(* IEC 61131-3 sources: AXOpen/src/showcase/app/src/ComponentsRexrothDrives/Documentation, 1 file *)

(* ---- Component_1.st ---- *)
USING AXOpen.Components.Abstractions.Drives;
USING AXOpen.Core;

NAMESPACE AXOpen.Components.Rexroth.Drives
    {S7.extern=ReadWrite}
    CLASS Component_1 EXTENDS AXOpen.Core.AxoObject
        //<ComponentDeclaration>
        VAR PUBLIC
            IndraDrive : AXOpen.Components.Rexroth.Drives.AxoIndraDrive;
        END_VAR
        //</ComponentDeclaration>

        //<InitializationArgumentsDeclaration>
        VAR PUBLIC
            manualControl   :   BOOL;
            Enable          :   BOOL;                       //  As long as ‘Enable’ is true, power is being enabled.
            EnablePositive  :   BOOL;                       //  As long as ‘Enable’ is true, this permits motion in positive direction
            EnableNegative  :   BOOL;                       //  As long as ‘Enable’ is true, this permits motion in negative direction
        END_VAR
        //</InitializationArgumentsDeclaration>

        METHOD PUBLIC OVERRIDE Run
            VAR_INPUT
                inParent : IAxoObject;
            END_VAR

            SUPER.Run(inParent);

            IF(manualControl) THEN
                IndraDrive.ActivateManualControl();
            END_IF;
            //<Initialization>
            IndraDrive.Run(inParent               :=  THIS,
                            hwID                :=  AXOpen.Showcase.HwIdentifiers#rexroth_indradrive_HwID,
                            Enable              :=  Enable,
                            EnablePositive      :=  EnablePositive,
                            EnableNegative      :=  EnableNegative);
            //</Initialization>

        THIS.UseInSequencer();
        END_METHOD

        //<Usage>
        VAR PUBLIC
            Sequencer : AxoSequencer;
            Steps : ARRAY[0..30] OF AXOpen.Core.AxoStep;
        END_VAR

        VAR PRIVATE
            _Valid : BOOL;
            _BoolValue  : BOOL;
            _DintValue  : DINT;
            _RealValue  : REAL;
            _i          : INT;
        END_VAR
        METHOD PRIVATE UseInSequencer

            Sequencer.Run(THIS);
            Sequencer.Open();
            Sequencer.SequenceMode := eAxoSequenceMode#RunOnce;

            _i := 0;
            IF(Steps[_i].Execute(Sequencer, 'Restore')) THEN
                manualControl := FALSE;
                Enable := FALSE;
                EnablePositive := FALSE;
                EnableNegative := FALSE;
                IndraDrive.Restore();
                Sequencer.MoveNext();
            END_IF;

            _i := _i + 1;
            IF(Steps[_i].Execute(Sequencer, 'Reset drive')) THEN
                IF(IndraDrive.AxoReset().IsDone()) THEN
                    Sequencer.MoveNext();
                END_IF;
            END_IF;

            _i := _i + 1;
            IF(Steps[_i].Execute(Sequencer, 'Enable drive')) THEN
                Enable := TRUE;
                EnablePositive := TRUE;
                EnableNegative := TRUE;
                IF(IndraDrive.AxoPower_Status) THEN
                    Sequencer.MoveNext();
                END_IF;
            END_IF;

            _i := _i + 1;
            IF(Steps[_i].Execute(Sequencer, 'Drive homming')) THEN
                IF(IndraDrive.AxoHome(  Position        :=  LREAL#5.0,
                                            HommingMode     :=  INT#551,
                                            Velocity        :=  LREAL#1.0,
                                            Acceleration    :=  LREAL#50.0,
                                            Deceleration    :=  LREAL#50.0
                                            ).IsDone()) THEN
                    IndraDrive.Restore();
                    Sequencer.MoveNext();
                END_IF;
            END_IF;

            _i := _i + 1;
            IF(Steps[_i].Execute(Sequencer, 'Check position')) THEN
                IF(IndraDrive.ActualPosition >=4.9 AND  IndraDrive.ActualPosition <=5.1) THEN
                    Sequencer.MoveNext();
                END_IF;
            END_IF;

            _i := _i + 1;
            IF(Steps[_i].Execute(Sequencer, 'Set position')) THEN
                IF(IndraDrive.AxoSetPosition(Position :=  LREAL#0.0).IsDone()) THEN
                    IndraDrive.Restore();
                    Sequencer.MoveNext();
                END_IF;
            END_IF;

            _i := _i + 1;
            IF(Steps[_i].Execute(Sequencer, 'Check position')) THEN
                IF(IndraDrive.ActualPosition >=-0.1 AND  IndraDrive.ActualPosition <=0.1) THEN
                    Sequencer.MoveNext();
                END_IF;
            END_IF;

            _i := _i + 1;
            IF(Steps[_i].Execute(Sequencer, 'Move absolute')) THEN
                IF(IndraDrive.AxoMoveAbsolute(  Position        :=  LREAL#5.0,
                                                    Velocity        :=  LREAL#10.0,
                                                    Acceleration    :=  LREAL#50.0,
                                                    Deceleration    :=  LREAL#50.0,
                                                    Jerk            :=  LREAL#50.0
                                                    ).IsDone()) THEN
                    IndraDrive.Restore();
                    Sequencer.MoveNext();
                END_IF;
            END_IF;

            _i := _i + 1;
            IF(Steps[_i].Execute(Sequencer, 'Check position')) THEN
                IF(IndraDrive.ActualPosition >=4.9 AND  IndraDrive.ActualPosition <=5.1) THEN
                    Sequencer.MoveNext();
                END_IF;
            END_IF;

            _i := _i + 1;
            IF(Steps[_i].Execute(Sequencer, 'Move additive')) THEN
                IndraDrive.AxoMoveAbsolute(  Position           :=  LREAL#10.0,
                                                    Velocity        :=  LREAL#1.0,
                                                    Acceleration    :=  LREAL#50.0,
                                                    Deceleration    :=  LREAL#50.0,
                                                    Jerk            :=  LREAL#50.0
                                                    );
                IF IndraDrive.ActualPosition > 7.5 THEN
                    IndraDrive.AxoMoveAdditive(  Distance        :=  LREAL#5.0,
                                                        Velocity        :=  LREAL#5.0,
                                                        Acceleration    :=  LREAL#50.0,
                                                        Deceleration    :=  LREAL#50.0,
                                                        Jerk            :=  LREAL#50.0
                                                        );
                END_IF;
                IF(IndraDrive.AxoMoveAdditive_Task.IsDone()) THEN
                    IndraDrive.Restore();
                    Sequencer.MoveNext();
                END_IF;
            END_IF;

            _i := _i + 1;
            IF(Steps[_i].Execute(Sequencer, 'Check position')) THEN
                IF(IndraDrive.ActualPosition >=14.9 AND  IndraDrive.ActualPosition <=15.1) THEN
                    Sequencer.MoveNext();
                END_IF;
            END_IF;

            _i := _i + 1;
            IF(Steps[_i].Execute(Sequencer, 'Move relative')) THEN
                IF(IndraDrive.AxoMoveRelative(  Distance        :=  LREAL#-5.0,
                                                    Velocity        :=  LREAL#10.0,
                                                    Acceleration    :=  LREAL#50.0,
                                                    Deceleration    :=  LREAL#50.0,
                                                    Jerk            :=  LREAL#50.0
                                                    ).IsDone()) THEN
                    IndraDrive.Restore();
                    Sequencer.MoveNext();
                END_IF;
            END_IF;

            _i := _i + 1;
            IF(Steps[_i].Execute(Sequencer, 'Check position')) THEN
                IF(IndraDrive.ActualPosition >=9.9 AND  IndraDrive.ActualPosition <=10.1) THEN
                    Sequencer.MoveNext();
                END_IF;
            END_IF;

            _i := _i + 1;
            IF(Steps[_i].Execute(Sequencer, 'Read digital input')) THEN
                IndraDrive.AxoReadDigitalInput(Enable := TRUE, InputNumber := 4 , Valid=> _Valid, Value => _BoolValue);
                IF(_Valid AND _BoolValue) THEN
                    IndraDrive.Restore();
                    Sequencer.MoveNext();
                    IndraDrive.AxoReadDigitalInput(Enable :=FALSE);
                END_IF;
            END_IF;

            _i := _i + 1;
            IF(Steps[_i].Execute(Sequencer, 'Move velocity')) THEN
                IndraDrive.AxoMoveVelocity(  Velocity        :=  LREAL#2.0,
                                                    Acceleration    :=  LREAL#50.0,
                                                    Deceleration    :=  LREAL#50.0,
                                                    Jerk            :=  LREAL#50.0,
                                                    Direction       :=  eAxoDriveDirection#NegativeDirection,
                                                    InVelocity      => _BoolValue);
                IF(_BoolValue) THEN
                    IndraDrive.Restore();
                    Sequencer.MoveNext();
                END_IF;
            END_IF;

            _i := _i + 1;
            IF(Steps[_i].Execute(Sequencer, 'Halt')) THEN
                IF(IndraDrive.AxoHalt(  Deceleration    :=  LREAL#50.0,
                                            Jerk            :=  LREAL#50.0
                                            ).IsDone()) THEN
                    IndraDrive.Restore();
                    Sequencer.MoveNext();
                END_IF;
            END_IF;

            _i := _i + 1;
            IF(Steps[_i].Execute(Sequencer, 'Move velocity')) THEN
                IndraDrive.AxoMoveVelocity(  Velocity        :=  LREAL#2.0,
                                                    Acceleration    :=  LREAL#50.0,
                                                    Deceleration    :=  LREAL#50.0,
                                                    Jerk            :=  LREAL#50.0,
                                                    Direction       :=  eAxoDriveDirection#NegativeDirection,
                                                    InVelocity      => _BoolValue);
                IF(_BoolValue) THEN
                    IndraDrive.Restore();
                    Sequencer.MoveNext();
                END_IF;
            END_IF;

            _i := _i + 1;
            IF(Steps[_i].Execute(Sequencer, 'Read digital input')) THEN
                IndraDrive.AxoReadDigitalInput(Enable := TRUE, InputNumber := 4 , Valid=> _Valid, Value => _BoolValue);
                IF(_Valid AND NOT _BoolValue) THEN
                    IndraDrive.Restore();
                    Sequencer.MoveNext();
                    IndraDrive.AxoReadDigitalInput(Enable :=FALSE);
                END_IF;
            END_IF;

            _i := _i + 1;
            IF(Steps[_i].Execute(Sequencer, 'Disable drive')) THEN
                Enable := FALSE;
                EnablePositive := TRUE;
                EnableNegative := TRUE;
                IF(NOT IndraDrive.AxoPower_Status) THEN
                    Sequencer.MoveNext();
                END_IF;
            END_IF;

            _i := _i + 1;
            IF(Steps[_i].Execute(Sequencer, 'Reset drive')) THEN
                IndraDrive.AxoReset();
                Sequencer.MoveNext();
            END_IF;

            _i := _i + 1;
            IF(Steps[_i].Execute(Sequencer, 'Enable drive')) THEN
                Enable := TRUE;
                EnablePositive := TRUE;
                EnableNegative := TRUE;
                IF(IndraDrive.AxoPower_Status) THEN
                    Sequencer.MoveNext();
                END_IF;
            END_IF;

            _i := _i + 1;
            IF(Steps[_i].Execute(Sequencer, 'Jog')) THEN
                manualControl := TRUE;
                IndraDrive.AxoJogPositive.RemoteSwitchOn := TRUE;
                IndraDrive.AxoJog_Velocity      :=  LREAL#1.0;
                IndraDrive.AxoJog_Acceleration  :=  LREAL#5.0;
                IndraDrive.AxoJog_Deceleration  :=  LREAL#5.0;
                IndraDrive.AxoJog_Jerk          :=  LREAL#10.0;
                IndraDrive.AxoJog_Direction     :=  AXOpen.Components.Abstractions.Drives.eAxoDriveDirection#PositiveDirection;

                IF(IndraDrive.ActualPosition > 0) THEN
                    Sequencer.MoveNext();
                    IndraDrive.AxoJogPositive.RemoteSwitchOn := FALSE;
                    manualControl := FALSE;
                END_IF;
            END_IF;

            _i := _i + 1;
            IF(Steps[_i].Execute(Sequencer, 'Torque control')) THEN
                IndraDrive.AxoTorqueControl(Torque          := LREAL#9.5 ,
                                                PositionLimit   :=  LREAL#100.0,
                                                Velocity        :=  LREAL#50.0,
                                                Acceleration    :=  LREAL#50.0,
                                                Deceleration    :=  LREAL#50.0,
                                                Jerk            :=  LREAL#50.0,
                                                Direction       :=  eAxoDriveDirection#PositiveDirection,
                                                InTorque      => _BoolValue);
                IF(_BoolValue) THEN
                    // IndraDrive.Restore();    removed due to we want to stay in torque up to reach the position 10.0
                    Sequencer.MoveNext();
                END_IF;
            END_IF;

            _i := _i + 1;
            IF(Steps[_i].Execute(Sequencer, 'Check position')) THEN
                IF(IndraDrive.ActualPosition >=10.0) THEN
                    IndraDrive.Restore(); // moved here from the prevous step
                    Sequencer.MoveNext();
                END_IF;
            END_IF;

            _i := _i + 1;
            IF(Steps[_i].Execute(Sequencer, 'Stop')) THEN
                IndraDrive.AxoStop(  Deceleration    :=  LREAL#50.0,
                                            Jerk            :=  LREAL#50.0,
                                            Done      => _BoolValue);
                IF(_BoolValue) THEN
                    Sequencer.MoveNext();
                END_IF;
            END_IF;

            _i := _i + 1;
            IF(Steps[_i].Execute(Sequencer, 'Release stop')) THEN
                IndraDrive.AxoStop_Task.Restore();
                IF(IndraDrive.AxoStop_Task.IsReady()) THEN
                    Sequencer.MoveNext();
                END_IF;
            END_IF;

            _i := _i + 1;
            IF(Steps[_i].Execute(Sequencer, 'Move absolute')) THEN
                IF(IndraDrive.AxoMoveAbsolute(  Position        :=  LREAL#0.0,
                                                    Velocity        :=  LREAL#50.0,
                                                    Acceleration    :=  LREAL#50.0,
                                                    Deceleration    :=  LREAL#50.0,
                                                    Jerk            :=  LREAL#50.0
                                                    ).IsDone()) THEN
                    IndraDrive.Restore();
                    Sequencer.MoveNext();
                END_IF;
            END_IF;

            _i := _i + 1;
            IF(Steps[_i].Execute(Sequencer, 'Disable drive')) THEN
                Enable := FALSE;
                EnablePositive := FALSE;
                EnableNegative := FALSE;
                IF(NOT IndraDrive.AxoPower_Status) THEN
                    Sequencer.MoveNext();
                END_IF;
            END_IF;

            _i := _i + 1;
            IF(Steps[_i].Execute(Sequencer, 'Reset drive')) THEN
                IF(IndraDrive.AxoReset().IsDone()) THEN
                    Sequencer.MoveNext();
                END_IF;
            END_IF;

            _i := _i + 1;
            IF(Steps[_i].Execute(Sequencer, 'Restore')) THEN
                IndraDrive.Restore();
                Sequencer.CompleteSequence();
            END_IF;
        END_METHOD
        //</Usage>
    END_CLASS
END_NAMESPACE
